{attribute 'qualified_only'}
VAR_GLOBAL
    tPassageOfTime      : TIME := TIME#0MS; // Keep track of the passage of time.
    eGlobalExampleEnum  : EXAMPLE_ENUM := EXAMPLE_ENUM.Example0;       // Global example ENUM
END_VAR

(* stored: Version 1.1.0.1, ProductVersion 3.1.4022.10
   GVL GVL: Id {e3330285-cffa-4779-85db-37f04fe46348} *)
